FUNCTION_BLOCK FbProblemTester EXTENDS TcUnit.FB_TestSuite
VAR
    _problem : IProblemSolver;
    _expectedResult : STRING;
END_VAR

TEST(TestName := '');
_problem.Execute := TRUE;
_problem.Cyclic();

IF _problem.Done THEN
    AssertEquals_STRING(Expected := _expectedResult, Actual := _problem.Result, Message := 'The problem solver did not return the correct answer.');
    _problem.Execute := FALSE;
    TEST_FINISHED();
END_IF

METHOD FB_init : BOOL
VAR_INPUT
    bInitRetains : BOOL; // if TRUE, the retain variables are initialized (warm start / cold start)
    bInCopyCode : BOOL; // if TRUE, the instance afterwards gets moved into the copy code (online change)
    problemSolver : IProblemSolver;
    expectedResult : STRING;
END_VAR
_problem := problemSolver;
_expectedResult := expectedResult;
END_METHOD

END_FUNCTION_BLOCK

(* stored: Version 1.1.0.1, ProductVersion 3.1.4024.9
   POU FbProblemTester: Id {8fc21e6d-9ed7-4dab-8911-6417cccd286f}, SpecialFunc None
   Method FB_init: Id {bda51afe-9882-4a88-8aab-be632de375b5} *)
